(* PLC project Unnamed, Unknown Unnamed 1 *)
(* stored: creationDateTime 2019-08-06T14:23:42, modificationDateTime 2021-09-10T14:17:04 *)

PROGRAM MainStuff
  VAR
    var0 : HMI_INT;
    var1 : HMI_INT;
  END_VAR

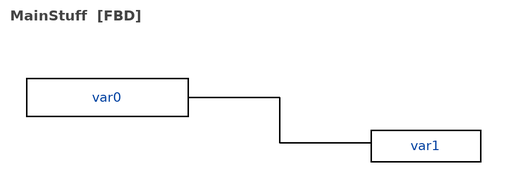
(* FBD diagram, written out as Structured Text *)
var1 := var0;
END_PROGRAM

CONFIGURATION config
  RESOURCE resource1 ON PLC
    TASK task0(INTERVAL := T#20ms, PRIORITY := 0);
    PROGRAM instance0 WITH task0 : MainStuff;
  END_RESOURCE
END_CONFIGURATION
